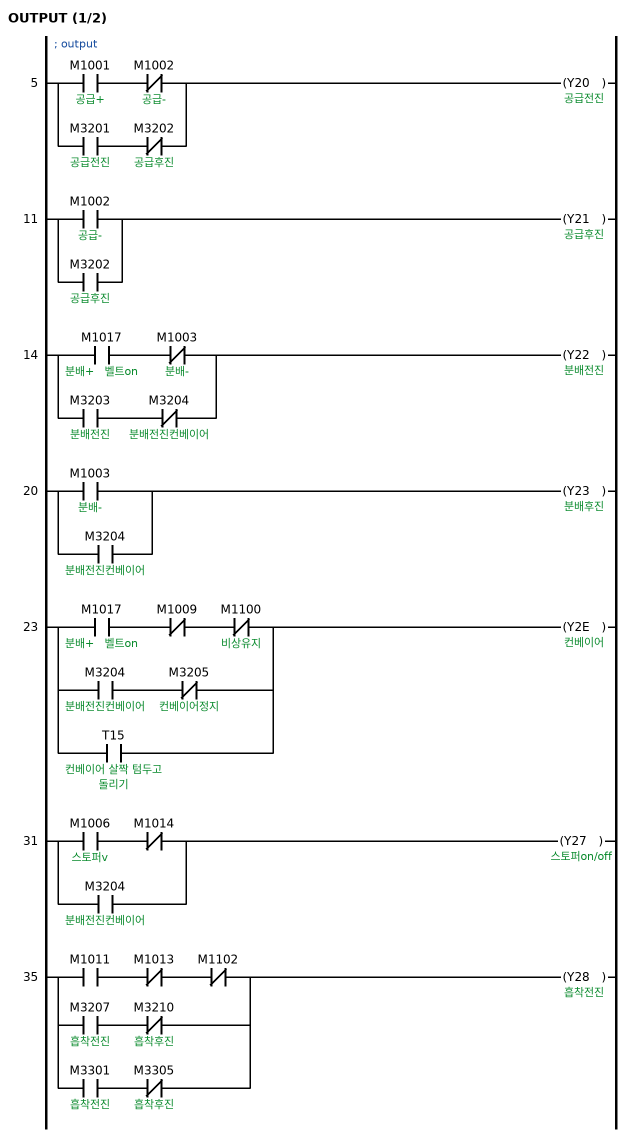
[picture p24: ladder of OUTPUT, rungs at steps 5 to 35]
; output
5     LD      M1001  ; 공급+
      ANI     M1002  ; 공급-
      LD      M3201  ; 공급전진
      ANI     M3202  ; 공급후진
      ORB
      OUT     Y20  ; 공급전진
11    LD      M1002  ; 공급-
      OR      M3202  ; 공급후진
      OUT     Y21  ; 공급후진
14    LD      M1017  ; 분배+   벨트on
      ANI     M1003  ; 분배-
      LD      M3203  ; 분배전진
      ANI     M3204  ; 분배전진컨베이어
      ORB
      OUT     Y22  ; 분배전진
20    LD      M1003  ; 분배-
      OR      M3204  ; 분배전진컨베이어
      OUT     Y23  ; 분배후진
23    LD      M1017  ; 분배+   벨트on
      ANI     M1009
      ANI     M1100  ; 비상유지
      LD      M3204  ; 분배전진컨베이어
      ANI     M3205  ; 컨베이어정지
      ORB
      OR      T15  ; 컨베이어 살짝 텀두고 돌리기
      OUT     Y2E  ; 컨베이어
31    LD      M1006  ; 스토퍼v
      ANI     M1014
      OR      M3204  ; 분배전진컨베이어
      OUT     Y27  ; 스토퍼on/off
35    LD      M1011
      ANI     M1013
      ANI     M1102
      LD      M3207  ; 흡착전진
      ANI     M3210  ; 흡착후진
      ORB
      LD      M3301  ; 흡착전진
      ANI     M3305  ; 흡착후진
      ORB
      OUT     Y28  ; 흡착전진
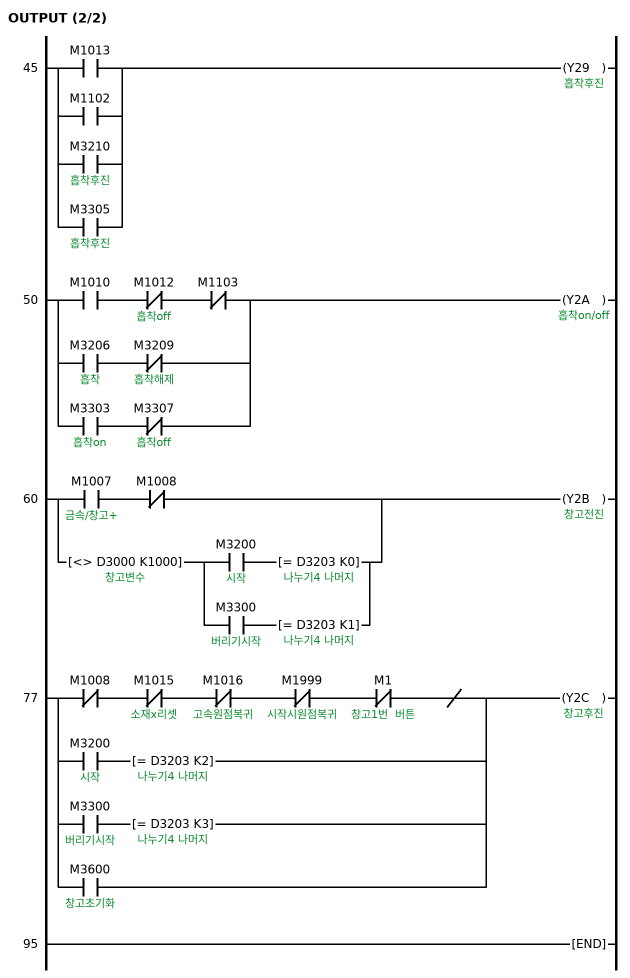
45    LD      M1013
      OR      M1102
      OR      M3210  ; 흡착후진
      OR      M3305  ; 흡착후진
      OUT     Y29  ; 흡착후진
50    LD      M1010
      ANI     M1012  ; 흡착off
      ANI     M1103
      LD      M3206  ; 흡착
      ANI     M3209  ; 흡착해제
      ORB
      LD      M3303  ; 흡착on
      ANI     M3307  ; 흡착off
      ORB
      OUT     Y2A  ; 흡착on/off
60    LD      M1007  ; 금속/창고+
      ANI     M1008
      LD<>    D3000 K1000  ; 창고변수
      LD      M3200  ; 시작
      AND=    D3203 K0  ; 나누기4 나머지
      LD      M3300  ; 버리기시작
      AND=    D3203 K1  ; 나누기4 나머지
      ORB
      ANB
      ORB
      OUT     Y2B  ; 창고전진
77    LDI     M1008
      ANI     M1015  ; 소재x리셋
      ANI     M1016  ; 고속원점복귀
      ANI     M1999  ; 시작시원점복귀
      ANI     M1  ; 창고1번  버튼
      INV
      LD      M3200  ; 시작
      AND=    D3203 K2  ; 나누기4 나머지
      ORB
      LD      M3300  ; 버리기시작
      AND=    D3203 K3  ; 나누기4 나머지
      ORB
      OR      M3600  ; 창고초기화
      OUT     Y2C  ; 창고후진
95    END
END_PROGRAM

// device comments not shown above
M102  ; 2번창고 적재
M103  ; 3번창고 적재
M104  ; 4번창고 적재
M202  ; 공급후진
M203  ; 분배전진
M204  ; 분배후진컨베이어
M205  ; 컨베이어정지
M206  ; 흡착
M207  ; 흡착전진
M208  ; 아래로 살짝내리기
M209  ; 흡착해제
M210  ; 흡착후진
M211  ; 초기위치로
M212  ; 끝
M300  ; 버리기 시작
M301  ; 흡착전진
M302  ; 살짝내리기
M303  ; 흡착on
M304  ; 살짝올리기
M305  ; 흡착후진
M306  ; 컨베이어로 내리기
M307  ; 흡착off
M308  ; 버리기  종료
M400  ; 끝나고 창고후진
M3402  ; 자기유지
M7998  ; ready
M7999  ; 원점확립
D102  ; zp값
D200  ; 나누기 몫
D201  ; 나머지
D202  ; 나누기 4 몫
D203  ; 나누기4 나머지
D3111  ; 나머지의나머지
